(* PLC project PlcMain, Beckhoff Automation GmbH TwinCAT PLC Control 3.5.13.21 *)
(* stored: creationDateTime 2022-08-19T12:32:47.6959428, modificationDateTime 2022-08-19T12:32:47.6959428 *)

{attribute 'qualified_only'}
{attribute 'strict'}
TYPE StateSeparator :
(
	Off,
	Init,
	Init_Wait,
	Ready,
	Eject,
	Eject_Wait_1,
	Eject_Wait_2,
	Done_Wait,
	Done
);
END_TYPE
